TYPE ST_VisionResult :
STRUCT
	bReady				: BOOL;
	bBusy				: BOOL;
	bResultValid		: BOOL;
	
	bPartPresent		: BOOL;
	bPartOK				: BOOL;
	
	nDefectCode			: UINT;
	
	fWidth          	: REAL;
    fHeight         	: REAL;
    fAngle          	: REAL;

    nProductID      	: DINT;	
END_STRUCT
END_TYPE

(* stored: Version 1.1.0.1, ProductVersion 3.1.4024.16
   DUT ST_VisionResult: Id {53ed8d9f-00fd-4541-b07c-c10f3587e1ae} *)
